Staubli VAL3: checkZone.pgx

program checkZone(point& x_pPoints[] (dimensions=1), tool x_tTool (dimensions=1), num x_nDimension (dimensions=1), num x_nType (dimensions=1), bool& x_bInside (dimensions=1))
begin
  // init the variable
  x_bInside=false
  // show the frame
  switch x_nType
    case 1
      //
      // BOX
      //
      //create the cube
      call solid:create_cube(x_pPoints[0],x_pPoints[1],x_pPoints[2],x_nDimension)
      // check the cube
      call solid:check_cube(x_tTool,x_bInside)
    break
    case 2
      //
      // SPHERE
      //
      // create the sphere
      call solid:create_sphere(x_pPoints,x_nDimension)
      // check the cube
      call solid:check_sphere(x_tTool,x_bInside)
    break
    case 3
      //
      // PLANE
      //
      //create the plane
      call solid:create_plane(x_pPoints[0],x_pPoints[1],x_pPoints[2])
      // check the cube
      call solid:check_plane(x_tTool,x_bInside)
    break
  endSwitch
end
